RoboDK station: TRABAJO PRACTICO 10.rdk

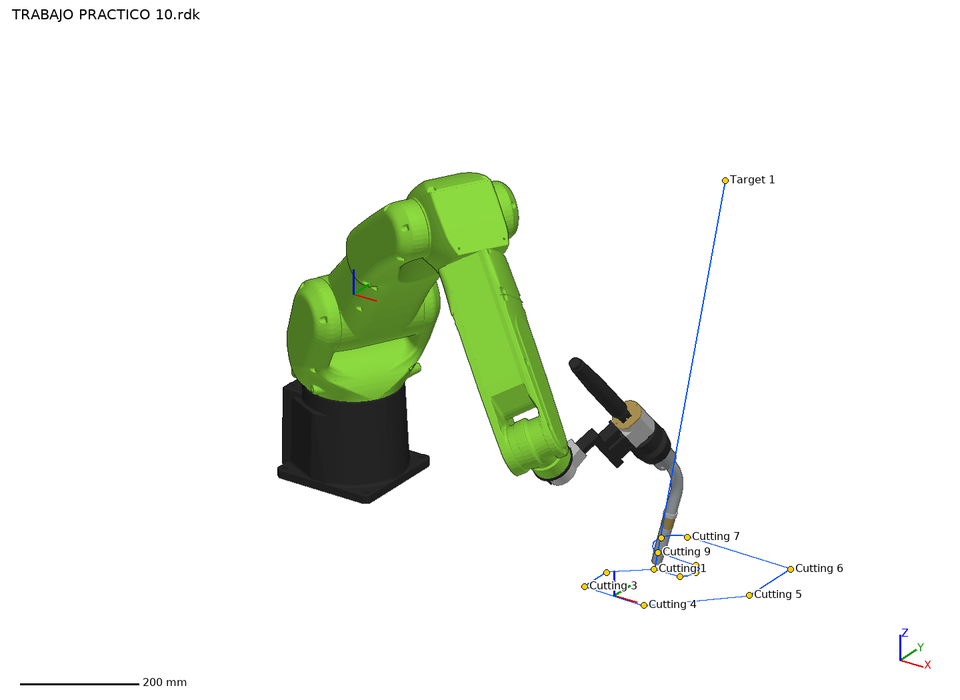
[picture v0: the station drawn from its stored meshes, robots at their saved joint values, targets as dots, program paths as lines]
Station 02 - Intro (saved by RoboDK 5.7.2). Poses are relative to the parent item; angles as X-Y-Z fixed-axis rotations.
  - frame Fanuc CR-7iA/L Base at (10, 0, 330) mm
    - robot Fanuc CR-7iA/L: 6 axes, payload 7 kg, reach 911 mm, repeatability 0.03 mm, weight 55 kg
        modified DH rows (alpha deg, a mm, theta deg, d mm): 0, 0, 0, 330; -90, 50, -90, 0; 0, 440, 0, 0; -90, 35, 0, 420; 90, 0, 0, 0; -90, 0, 0, 80
        base shift (0, 0, -330) mm
        joint limits [-170, -100, -67, -190, -115, -360] to [170, 145, 213, 190, 115, 360]; home [0, 0, 0, 0, 0, 0]; saved at [-29.091, 46.974, -44.756, 140.36, 70.717, -70.984]
      - tool OTC Daihen FD-84 Welding Gun, TCP at (0, 0, 400) mm, rotated rx 0 ry -80 rz 0 deg, size 201.6 x 65.1 x 567.7 mm
    - frame Part at (634.18, -140.58, -330) mm
      - object Cutting sheet at (-60, 0, 0) mm, size 250 x 250 x 3 mm, geometry from Cutting sheet.STEP
      - target Target 1 (Cartesian target) at (77.1, 213.72, 711.99) mm, rotated rx -170.17 ry -17.05 rz 38.65 deg; joints [-34.031, -4.501, -20.845, 77.493, 78.178, -76.339] of Fanuc CR-7iA/L
      - target Cutting 1 (Cartesian target) at (-3.03, 120.17, 0) mm, rotated rx -156.33 ry 39.46 rz 79.6 deg; joints [-29.091, 46.974, -44.756, -39.64, -70.717, -250.984] of Fanuc CR-7iA/L
      - target Cutting 2 (Cartesian target) at (-59.16, 60.84, 2.01) mm, rotated rx 54.74 ry 30 rz -9.74 deg; joints [20.833, 65.664, -136.473, -36.701, 103.422, -258.976] of Fanuc CR-7iA/L
      - target Cutting 3 (Cartesian target) at (-61.13, -0.64, 0) mm, rotated rx 180 ry 45 rz 79.6 deg; joints [-38.212, 41.286, -44.15, -33.239, -67.754, -223.29] of Fanuc CR-7iA/L
      - target Cutting 4 (Cartesian target) at (61.85, -2.92, 0) mm, rotated rx 180 ry 45 rz 79.6 deg; joints [-32.66, 52.524, -33.793, -33.514, -74.034, -233.13] of Fanuc CR-7iA/L
      - target Cutting 5 (Cartesian target) at (189.07, 124.37, 3) mm, rotated rx -180 ry 45 rz 79.6 deg; joints [-20.356, 60.252, -25.923, -35.913, -74.399, -246.888] of Fanuc CR-7iA/L
      - target Cutting 6 (Cartesian target) at (187.92, 246.72, 3) mm, rotated rx 180 ry 45 rz 79.6 deg; joints [-12.033, 55.162, -30.825, -38.851, -66.062, -249.912] of Fanuc CR-7iA/L
      - target Cutting 7 (Cartesian target) at (-24.67, 249.16, 3) mm, rotated rx 180 ry 45 rz 79.6 deg; joints [-16.16, 33.005, -50.692, -45.366, -53.318, -231.808] of Fanuc CR-7iA/L
      - target Cutting 8 (Cartesian target) at (-59.3, 221.28, 3) mm, rotated rx 180 ry 45 rz 79.6 deg; joints [-19.898, 30.763, -52.498, -44.597, -53.682, -228.177] of Fanuc CR-7iA/L
      - target Cutting 9 (Cartesian target) at (-31, 172.19, 3) mm, rotated rx -180 ry 45 rz 79.6 deg; joints [-23.372, 34.888, -49.135, -41.432, -57.638, -229.011] of Fanuc CR-7iA/L
      - target Cutting 10 (Cartesian target) at (48.85, 168.65, 3) mm, rotated rx 180 ry 45 rz 79.6 deg; joints [-20.969, 42.281, -42.741, -39.957, -61.399, -235.318] of Fanuc CR-7iA/L
      - target Cutting 11 (Cartesian target) at (65.48, 144.75, 3) mm, rotated rx 180 ry 45 rz 79.6 deg; joints [-22.304, 44.828, -40.452, -38.719, -63.803, -236.083] of Fanuc CR-7iA/L
      - target Cutting 12 (Cartesian target) at (48.36, 121.91, 0) mm, rotated rx 180 ry 45 rz 79.6 deg; joints [-24.58, 44.358, -41.384, -38.169, -64.142, -233.939] of Fanuc CR-7iA/L
  - object Table 1200x1000mm (Welding) at (410, 0, 0) mm, size 1193.8 x 965.2 x 609.6 mm, geometry from Table-1200x1000mm-Welding.sld
  - program Prog1 (14 instructions, listed below)
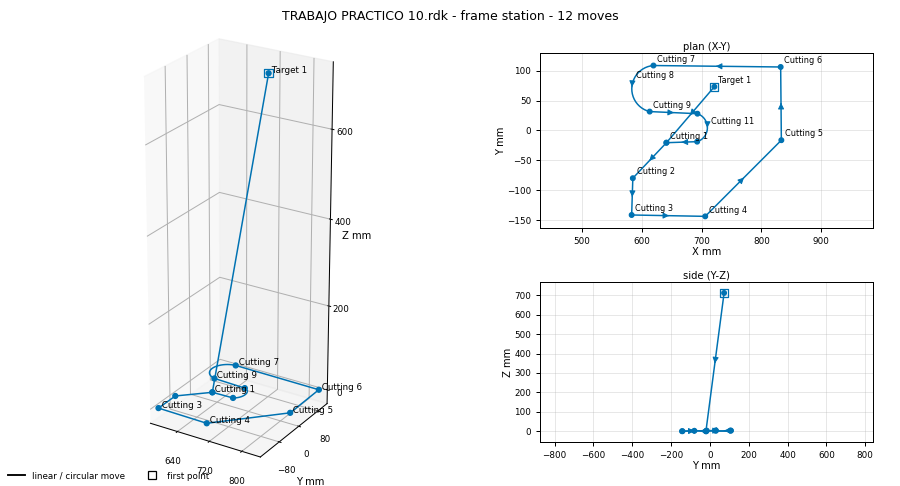
[picture p0: tool path of TRABAJO PRACTICO 10.rdk in frame station, 12 of 12 moves have a stored position in this frame; points joined in program order, loops and branches not executed]

--- program Prog1 (robot Fanuc CR-7iA/L) ---
  Est. Ref.: Part
  Est. herr: OTC Daihen FD-84 Welding Gun
  MoveJ (Target 1)
  MoveL (Cutting 1)
  MoveL (Cutting 2)
  MoveL (Cutting 3)
  MoveL (Cutting 4)
  MoveL (Cutting 5)
  MoveL (Cutting 6)
  MoveL (Cutting 7)
  MoveC (Cutting 8, Cutting 11) -> target Cutting 9
  MoveL (Cutting 12) -> target Cutting 10
  MoveC (Cutting 13, Cutting 14) -> target Cutting 11 -> target Cutting 12
  MoveL (Cutting 1)
